SYSTEM SystemTrafficLightIcaru2 (* System Configuration *)
  (* Standard: 61499-1 *)
  (* Version 0.4, 2009-03-05, JHC, Holobloc Inc., Deleted Application. *)
  (* Version 0.3, 2003-12-05, JHC, Rockwell Automation, Renamed from NEWSYSTEM. *)
  (* Version 0.2, 2002-11-05, JHC, Rockwell Automation, Fixed missing (empty) FBD in Application. *)
  (* Version 0.1, 2002-01-17, JHC, Rockwell Automation, Minor cleanup *)
  (* Version 0.0, 2000-05-27, JHC, Rockwell Automation *)
  DEVICE DEV_CONTROL : FRAME_DEVICE(BOUNDS := [100,100,150,200], GRID := [1,4])
    RESOURCE RES2 : PANEL_RESOURCE(ROWS := 4)
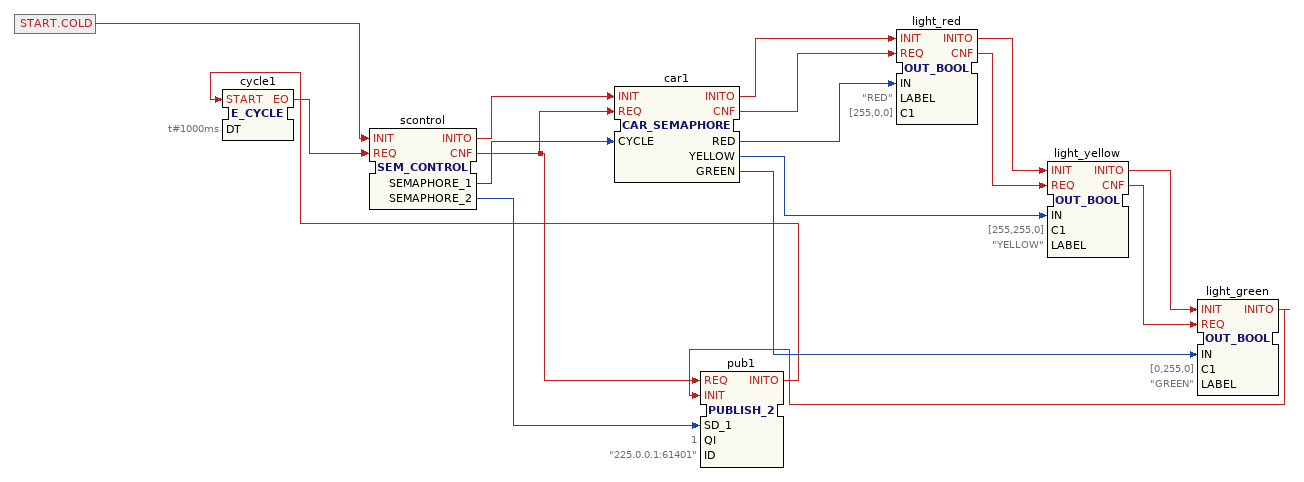
      FBS
        scontrol : SEM_CONTROL;
        cycle1 : E_CYCLE(DT := t#1000ms);
        car1 : CAR_SEMAPHORE;
        light_red : OUT_BOOL(LABEL := "RED", C1 := [255,0,0]);
        light_yellow : OUT_BOOL(C1 := [255,255,0], LABEL := "YELLOW");
        light_green : OUT_BOOL(C1 := [0,255,0], LABEL := "GREEN");
        pub1 : PUBLISH_2(QI := 1, ID := "225.0.0.1:61401");
      END_FBS
      EVENT_CONNECTIONS
        START.COLD TO scontrol.INIT;
        light_red.INITO TO light_yellow.INIT;
        light_yellow.INITO TO light_green.INIT;
        light_red.CNF TO light_yellow.REQ;
        light_yellow.CNF TO light_green.REQ;
        scontrol.INITO TO car1.INIT;
        car1.INITO TO light_red.INIT;
        car1.CNF TO light_red.REQ;
        scontrol.CNF TO car1.REQ;
        cycle1.EO TO scontrol.REQ;
        scontrol.CNF TO pub1.REQ;
        light_green.INITO TO pub1.INIT;
        pub1.INITO TO cycle1.START;
      END_CONNECTIONS
      DATA_CONNECTIONS
        scontrol.SEMAPHORE_1 TO car1.CYCLE;
        car1.RED TO light_red.IN;
        car1.YELLOW TO light_yellow.IN;
        car1.GREEN TO light_green.IN;
        scontrol.SEMAPHORE_2 TO pub1.SD_1;
      END_CONNECTIONS
    END_RESOURCE
  END_DEVICE
  DEVICE DEV_SLAVE : DEV_ICARU_PC
    RESOURCE RES1 : ICARU_RES2
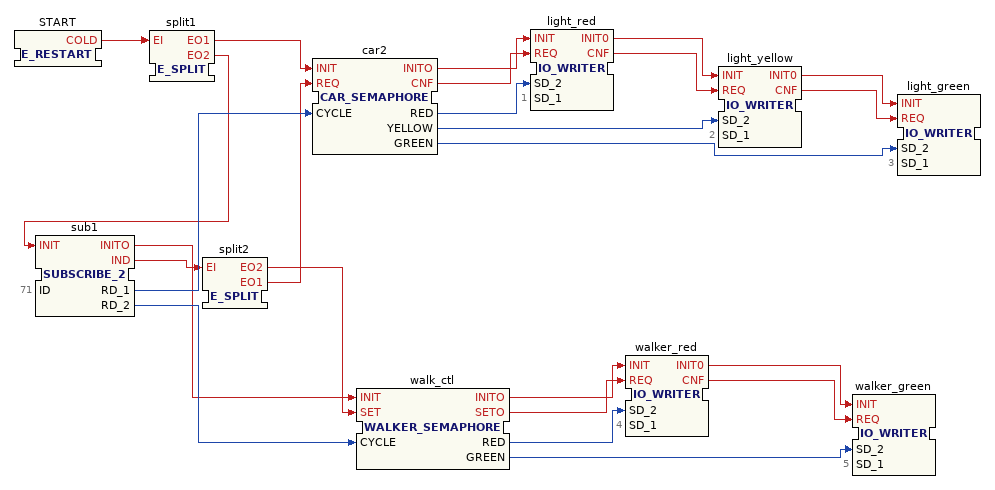
      FBS
        START : E_RESTART;
        car2 : CAR_SEMAPHORE;
        walk_ctl : WALKER_SEMAPHORE;
        sub1 : SUBSCRIBE_2(ID := 71);
        light_red : IO_WRITER(SD_1 := 1);
        light_yellow : IO_WRITER(SD_1 := 2);
        light_green : IO_WRITER(SD_1 := 3);
        walker_red : IO_WRITER(SD_1 := 4);
        walker_green : IO_WRITER(SD_1 := 5);
        split1 : E_SPLIT;
        split2 : E_SPLIT;
      END_FBS
      EVENT_CONNECTIONS
        sub1.INITO TO walk_ctl.INIT;
        light_red.INIT0 TO light_yellow.INIT;
        light_yellow.INIT0 TO light_green.INIT;
        walk_ctl.INITO TO walker_red.INIT;
        walker_red.INIT0 TO walker_green.INIT;
        walk_ctl.SETO TO walker_red.REQ;
        light_red.CNF TO light_yellow.REQ;
        light_yellow.CNF TO light_green.REQ;
        walker_red.CNF TO walker_green.REQ;
        START.COLD TO split1.EI;
        split1.EO1 TO car2.INIT;
        split1.EO2 TO sub1.INIT;
        sub1.IND TO split2.EI;
        split2.EO2 TO walk_ctl.SET;
        car2.INITO TO light_red.INIT;
        split2.EO1 TO car2.REQ;
        car2.CNF TO light_red.REQ;
      END_CONNECTIONS
      DATA_CONNECTIONS
        sub1.RD_1 TO car2.CYCLE;
        sub1.RD_2 TO walk_ctl.CYCLE;
        car2.RED TO light_red.SD_2;
        car2.YELLOW TO light_yellow.SD_2;
        car2.GREEN TO light_green.SD_2;
        walk_ctl.RED TO walker_red.SD_2;
        walk_ctl.GREEN TO walker_green.SD_2;
      END_CONNECTIONS
    END_RESOURCE
  END_DEVICE
END_SYSTEM
